// TIA Portal V17 export
// export: Created 2024-08-20T13:26:11.091301Z, ExportSetting WithDefaults, DisplayName Totally Integrated Automation Portal, DisplayVersion V17 Update 4, DisplayName TIA Portal Openness, DisplayVersion V17 Update 4, DisplayName TIA Portal Version Control Interface, DisplayVersion V17, DisplayName STEP 7 Professional, DisplayVersion V17 Update 4, DisplayName STEP 7 Safety, DisplayVersion V17, DisplayName WinCC Advanced, DisplayVersion V17 Update 4
DATA_BLOCK "VARIAVEIS"   // DB304
{ S7_Optimized_Access := 'FALSE' }
VERSION : 0.1
// stored: AutoNumber false, DBAccessibleFromOPCUA true, IsOnlyStoredInLoadMemory false, IsWriteProtectedInAS false
   VAR
      "MB-01-YST" : Real;   // Frequência raspador de areia
      "MB-01-YIT" : Real;   // Corrente raspador de areia
      "MB-02-YIT" : Real;   // Corrente raspador de areia
      "MB-02-YST" : Real;   // Frequência raspador de areia
      "MB-03-YIT" : Real;   // Corrente raspador de areia
      "MB-03-YST" : Real;   // Frequência raspador de areia
      "MB-04-YIT" : Real;   // Corrente raspador de areia
      "MB-04-YST" : Real;   // Frequência raspador de areia
      LIT_001 : Real;   // Nível Tanque
      "LIT_001-P" : Real;   // Percentual Tanque
      "PCM-E-CF-01-04-P100-ETRS" : Real;   // Tensão entre fases R e S
      "PCM-E-CF-01-04-P100-ETST" : Real;   // Tensão entre fases S e T
      "PCM-E-CF-01-04-P100-ETTR" : Real;   // Tensão entre fases T e R
      "PCM-E-CF-01-04-P100-ITR" : Real;   // Corrente fase R
      "PCM-E-CF-01-04-P100-ITS" : Real;   // Corrente fase S
      "PCM-E-CF-01-04-P100-ITT" : Real;   // Corrente fase T
      "PCM-E-CF-01-04-P100-JPT" : Real;   // Potência ativa total
      "PCM-E-CF-01-04-P100-JQT" : Real;   // Potência reativa total
      "PCM-E-CF-01-04-P100-JST" : Real;   // Potência aparente total
      "PCM-E-CF-01-04-P100-FP" : Real;   // Fator de potência
      "QGBT-AUX-01-P100-ETRS" : Real;   // Tensão entre fases R e S
      "QGBT-AUX-01-P100-ETST" : Real;   // Tensão entre fases S e T
      "QGBT-AUX-01-P100-ETTR" : Real;   // Tensão entre fases T e R
      "QGBT-AUX-01-P100-ITR" : Real;   // Corrente fase R
      "QGBT-AUX-01-P100-ITS" : Real;   // Corrente fase S
      "QGBT-AUX-01-P100-ITT" : Real;   // Corrente fase T
      "QGBT-AUX-01-P100-JPT" : Real;   // Potência ativa total
      "QGBT-AUX-01-P100-JQT" : Real;   // Potência reativa total
      "QGBT-AUX-01-P100-JST" : Real;   // Potência aparente total
      "QGBT-AUX-01-P100-FP" : Real;   // Fator de potência
   END_VAR
BEGIN
END_DATA_BLOCK
